// TIA Portal V19 export
DATA_BLOCK "INPUT MAPING DB"   // DB1
{ S7_Optimized_Access := 'FALSE' }
   VAR
      "CIP RUN" : Bool;
      "SPARE(1)" : Bool;
      "SPARE(2)" : Bool;
      "P-201 A RO 1 FEED PUMP TRIP" : Bool;
      "P-201 B RO 1 FEED PUMP TRIP" : Bool;
      "P-201 C RO 1 FEED PUMP TRIP" : Bool;
      "P-301 A RO 1 HPP PUMP TRIP" : Bool;
      "P-301 B RO B HPP PUMP TRIP" : Bool;
      "P-401 A RO 2 FEED PUMP TRIP" : Bool;
      "P-401 B RO 2 FEED PUMP TRIP" : Bool;
      "P-401 C RO 2 FEED PUMP TRIP" : Bool;
      "P 401 A RO 2 HPP PUMP TRIP" : Bool;
      "P-401 B RO 2 HPP PUMP TRIP" : Bool;
      "LPS 301 RO 1" : Bool;
      "HPS-301 RO 1 PRESSURE SWITCH" : Bool;
      "LPS-302 RO 1 PRESSURE SWITCH" : Bool;
      "HPS-302 RO 1 PRESSURE SWITCH" : Bool;
      "LPS-401 RO 2 PRESSURE SWITCH" : Bool;
      "HPS-401 RO 2 PRESSURE SWITCH" : Bool;
      "LPS-402 RO 2 PRESSURE SWITCH" : Bool;
      "HPS-402 RO 2 PRESSURE SWITCH" : Bool;
      "DP-703 RO 1 DOSER LEVEL SWITCH" : Bool;
      "DP-704 RO 1 DOSER LEVEL SWITCH" : Bool;
      "DP-705 RO 1 DOSER LEVEL SWITCH" : Bool;
      "P-501 A EDI FEED PUMP TRIP" : Bool;
      "P-501 B EDI FEED PUMP TRIP" : Bool;
      "P-501 C EDI FEED PUMP TRIP" : Bool;
      "EDI 501 A TRIP" : Bool;
      "EDI 501 B TRIP" : Bool;
      "SPARE(8)" : Bool;
      "P-201 A RO 1 FEED PUMP FEED BACK" : Bool;
      "P-201 B RO 1 FEED PUMP FEED BACK" : Bool;
      "P-201 C RO 1 FEED PUMP FEED BACK" : Bool;
      "P-301 A RO 1 HPP PUMP FEED BACK" : Bool;
      "P-301 B RO 1 HPP PUMP FEED BACK" : Bool;
      "P-401 A R0 2 FEED PUMP FEED BACK" : Bool;
      "P-401 B RO 2 FEED PUMP FEED BACK" : Bool;
      "P-401 C RO 2 FEED PUMP FEED BACK" : Bool;
      "P-402 A RO 2 HPP PUMP FEED BACK" : Bool;
      "P-402 B RO 2 HPP PUMP FEED BACK" : Bool;
      "P-501 A EDI FEED PUMP FEED BACK" : Bool;
      "P-501 B EDI FEED PUMP FEED BACK" : Bool;
      "P-501 C EDI FEED PUMP FEED BACK" : Bool;
      "SPARE(3)" : Bool;
      "ABFV-301 FEED BACK OPEN" : Bool;
      "ABFV-301 FEED BACK CLOSE" : Bool;
      "ABFV-302 OPEN FEED BACK" : Bool;
      "ABFV-302 CLOSE FEED BACK" : Bool;
      "AGLV-301 OPEN FEED BACK" : Bool;
      "AGLV-301 CLOSE FEED BACK" : Bool;
      "AGLV-302 OPEN FEED BACK" : Bool;
      "AGLV-302 CLOSE FEED BACK" : Bool;
      "AGLV-401 OPEN FEED BACK" : Bool;
      "AGLV-401 CLOSE FEED BACK" : Bool;
      "AGLV-402 OPEN FEED BACK" : Bool;
      "AGLV-402 CLOSE FEED BACK" : Bool;
      "AGLV-501OPEN FEED BACK" : Bool;
      "AGLV-501 CLOSE FEED BACK" : Bool;
      "AGLV-502 OPEN FEED BACK" : Bool;
      "AGLV-502 CLOSE FEED BACK" : Bool;
      "SPARE(4)" : Bool;
      "SPARE(5)" : Bool;
   END_VAR
BEGIN
END_DATA_BLOCK
